{attribute 'linkalways'} 
{attribute 'no_explicit_call' := 'This FB is a CLASS and must be accessed using methods or properties'}
{attribute 'enable_dynamic_creation'}
FUNCTION_BLOCK Node_F_VN_ImageAbsoluteAverage EXTENDS VisionNode
VAR
    ipSrcImage : _ITcVnImage;
    fAverage : _LREAL(0.0);
    hrPrev : _HRESULT(S_OK);
	hresult : _HRESULT(S_OK);
END_VAR

METHOD PUBLIC  Clone : I_Node
VAR
	pNode : POINTER TO Node_F_VN_ImageAbsoluteAverage;
END_VAR
pNode := __NEW(Node_F_VN_ImageAbsoluteAverage);
Clone := pNode^;
END_METHOD

METHOD FB_init : BOOL
VAR_INPUT
	bInitRetains : BOOL; // if TRUE, the retain variables are initialized (warm start / cold start)
	bInCopyCode : BOOL;  // if TRUE, the instance afterwards gets moved into the copy code (online change)
END_VAR
AddInput('ipSrcImage', ipSrcImage);
AddInput('hrPrev', hrPrev);
AddOutput('fAverage', fAverage);
AddOutput('hresult', hresult);
END_METHOD

METHOD PROTECTED OnExecute
hresult.Value := F_VN_ImageAbsoluteAverage(
	ipSrcImage := ipSrcImage.Value,
    fAverage := fAverage.Value,
	hrPrev:= hrPrev.Value);
END_METHOD

METHOD PUBLIC PreExecutionCheck
VAR_INPUT
	Check : I_PreExecutionChecks;
END_VAR
Check.IsTrue(ipSrcImage.IsValid, 'ipSrcImage must contain an image');
END_METHOD

END_FUNCTION_BLOCK

(* stored: Version 1.1.0.1, ProductVersion 3.1.4024.13
   POU Node_F_VN_ImageAbsoluteAverage: Id {d29d625a-5e63-095b-227b-fc6b9a9d3d2e}, SpecialFunc None
   Folder Constructor: Id {a84ce2fe-560b-0226-38ee-b14c6931a549}
   Method Clone: Id {ff493f6f-1774-0881-2716-fd36ef086989}
   Method FB_init: Id {e94bce1e-f6df-0de7-1770-6bcf12985011}
   Method OnExecute: Id {c7bea972-74dd-0a75-3e1e-c99afceb048e}
   Method PreExecutionCheck: Id {e56d624d-afad-0867-24a9-43b42784d7f9} *)
